(* TLS/PSK configuration *)
{attribute 'no_explicit_call':='Direct call not allowed for type FB_TlsConfig'}
{attribute 'no_assign'}
FUNCTION_BLOCK FB_TlsConfig
VAR
	_pskKey       : ARRAY[0..TCPADS_TLS_MAX_PSK_KEY_SIZE] OF BYTE;
	_pskKeyLen    : UDINT:=0;
	_sIdentity    : STRING(TCPADS_TLS_PSK_IDENTITY_SIZE);
	_sCaPath      : STRING(TCPADS_TLS_CERTIFICATE_PATH_SIZE);
	_sCrlPath     : STRING(TCPADS_TLS_CERTIFICATE_PATH_SIZE);
	_sCertPath    : STRING(TCPADS_TLS_CERTIFICATE_PATH_SIZE);
	_sKeyPath     : STRING(TCPADS_TLS_CERTIFICATE_PATH_SIZE);
	_sKeyPwd      : STRING(TCPADS_TLS_KEY_PASSWORD_SIZE);
	_listenFlags  : ST_TlsListenFlags:=DEFAULT_TLSLISTENFLAGS;
	_connectFlags : ST_TlsConnectFlags:=DEFAULT_TLSCONNECTFLAGS;
END_VAR

(* Adds CA certificate path *)
METHOD FINAL AddCa
VAR_INPUT
	sCaPath : STRING(TCPADS_TLS_CERTIFICATE_PATH_SIZE);
END_VAR
_sCaPath:=sCaPath;
END_METHOD

(* Adds certificate path *)
METHOD FINAL AddCert
VAR_INPUT
	sCertPath: STRING(TCPADS_TLS_CERTIFICATE_PATH_SIZE);
	sKeyPath: STRING(TCPADS_TLS_CERTIFICATE_PATH_SIZE);
	sKeyPwd: STRING(TCPADS_TLS_KEY_PASSWORD_SIZE);
END_VAR
_sCertPath:=sCertPath;
_sKeyPath:=sKeyPath;
_sKeyPwd:=sKeyPwd;
END_METHOD

METHOD FINAL AddConnectFlags
VAR_INPUT
	flags : ST_TlsConnectFlags;
END_VAR
_connectFlags:=flags;
END_METHOD

(* Adds certificate revocation list path *)
METHOD FINAL AddCrl
VAR_INPUT
	sCrlPath : STRING(TCPADS_TLS_CERTIFICATE_PATH_SIZE);
END_VAR
_sCrlPath:=sCrlPath;
END_METHOD

METHOD FINAL AddListenFlags
VAR_INPUT
	flags : ST_TlsListenFlags;
END_VAR
_listenFlags:=flags;
END_METHOD

(* Adds PSK and PSK identity *)
METHOD FINAL AddPsk
VAR_IN_OUT
	key : ARRAY[*] OF BYTE;
END_VAR
VAR_INPUT
	sIdentity : STRING(TCPADS_TLS_PSK_IDENTITY_SIZE);
END_VAR
_pskKeyLen:=MIN(DINT_TO_UDINT(UPPER_BOUND(key, 1) - LOWER_BOUND(key, 1) + 1), TCPADS_TLS_MAX_PSK_KEY_SIZE, SIZEOF(_pskKey));
MEMCPY(ADR(_pskKey[0]), ADR(key[LOWER_BOUND(key, 1)]), _pskKeyLen);
_sIdentity:=sIdentity;
END_METHOD

METHOD FINAL Clear
_sIdentity:='';
_pskKeyLen:=0;
MEMSET(ADR(_pskKey[0]), 0, SIZEOF(_pskKey));
_sCaPath:='';
_sCertPath:='';
_sKeyPath:='';
_sKeyPwd:='';
_sCrlPath:='';
_listenFlags:=DEFAULT_TLSLISTENFLAGS;
_connectFlags:=DEFAULT_TLSCONNECTFLAGS;
END_METHOD

PROPERTY FINAL connectFlags : ST_TlsConnectFlags
GET
connectFlags:=_connectFlags;
END_GET
END_PROPERTY

PROPERTY FINAL listenFlags : ST_TlsListenFlags
GET
listenFlags:=_listenFlags;
END_GET
END_PROPERTY

(* Pointer to first PSK key byte *)
PROPERTY FINAL pskKey : PVOID
GET
pskKey:=SEL(_pskKeyLen = 0, ADR(_pskKey[0]), 0);
END_GET
END_PROPERTY

(* Byte size of PSK key *)
PROPERTY FINAL pskKeyLen : UDINT(0..TCPADS_TLS_MAX_PSK_KEY_SIZE)
GET
pskKeyLen:=_pskKeyLen;
END_GET
END_PROPERTY

(* CA certificate path *)
PROPERTY FINAL sCaPath : STRING(TCPADS_TLS_CERTIFICATE_PATH_SIZE)
GET
sCaPath:=_sCaPath;
END_GET
END_PROPERTY

(* Certificate path *)
PROPERTY FINAL sCertPath : STRING(TCPADS_TLS_CERTIFICATE_PATH_SIZE)
GET
sCertPath:=_sCertPath;
END_GET
END_PROPERTY

(* Certificate revocation list path *)
PROPERTY FINAL sCrlPath : STRING(TCPADS_TLS_CERTIFICATE_PATH_SIZE)
GET
sCrlPath:=_sCrlPath;
END_GET
END_PROPERTY

(* PSK key identity *)
PROPERTY FINAL sIdentity : STRING(TCPADS_TLS_PSK_IDENTITY_SIZE)
GET
sIdentity:=_sIdentity;
END_GET
END_PROPERTY

(* Certificate key path *)
PROPERTY FINAL sKeyPath : STRING(TCPADS_TLS_CERTIFICATE_PATH_SIZE)
GET
sKeyPath:=_sKeyPath;
END_GET
END_PROPERTY

(* Certificate key password *)
PROPERTY FINAL sKeyPwd : STRING(TCPADS_TLS_KEY_PASSWORD_SIZE)
GET
sKeyPwd:=_sKeyPwd;
END_GET
END_PROPERTY

END_FUNCTION_BLOCK

(* stored: Version 1.1.0.1
   POU FB_TlsConfig: Id {93bcd84a-f561-4920-9d01-802eb4450dac}, SpecialFunc None
   Method AddCa: Id {4d8dd57f-2b76-460c-be32-e417cbfae496}
   Method AddCert: Id {7460eebe-2dbe-400d-b22e-78f8c448e3cb}
   Method AddConnectFlags: Id {926e4460-d1ff-4890-afe0-63153b70e046}
   Method AddCrl: Id {de1979dc-ce82-460a-a963-c1dc8cbe1ced}
   Method AddListenFlags: Id {872e0c38-6839-4efd-affd-f4e34eab9833}
   Method AddPsk: Id {c23e5f48-6938-42d7-bd49-6a2527cefc0f}
   Method Clear: Id {2fcc3a28-c012-4bfa-8dd5-5117b18873f0}
   Property connectFlags: Id {d5ac45f6-4175-46d2-80a7-5d97502fcb40}
   Get Get: Id {a6df7a83-1dac-4c0c-8d86-d2e6d73344d6}
   Property listenFlags: Id {56b43e47-5dbf-4d79-90cc-0adddcfc7947}
   Get Get: Id {8e3a63f5-4283-4ad0-9198-ad2604cbb062}
   Property pskKey: Id {6f5939d6-f54a-47e1-b64f-1c244290a454}
   Get Get: Id {a07559dd-a5f0-4838-ab33-8ee0fc7236c0}
   Property pskKeyLen: Id {854c238a-2ee8-45ee-9d22-eca68074b39f}
   Get Get: Id {46a5fe42-42d2-486a-bb6d-b866c6724fd3}
   Property sCaPath: Id {31c41dec-4783-462c-b132-79bd87e6ca73}
   Get Get: Id {e6f02541-0d17-4f2b-8e3d-7b5e96c9d274}
   Property sCertPath: Id {a472a82e-f737-4230-9981-76b233e002fd}
   Get Get: Id {342c70b2-3518-470f-8ce1-0ad4d434e5c1}
   Property sCrlPath: Id {c25655e6-7a93-403f-8b12-966fee565163}
   Get Get: Id {6f63d266-2245-44ea-b92f-bfd8efd0f05b}
   Property sIdentity: Id {576713a3-8944-47d7-90b9-ca8ef1f97364}
   Get Get: Id {a074f4a3-9ed8-4836-b2f0-891e8e69a4f0}
   Property sKeyPath: Id {9d42f7d7-3ac1-4045-b668-9cf70f4bf8c2}
   Get Get: Id {30d4490f-0168-4cb6-8fe2-7be151c9fc17}
   Property sKeyPwd: Id {94695904-186a-4fe3-9764-cfa31177cce9}
   Get Get: Id {bf39b217-0b4c-45d5-ad3e-5da57f138972} *)
